FUNCTION_BLOCK FB_MachineControl EXTENDS FB_UniversalMachine IMPLEMENTS I_MachineControl
VAR
	(* Auxilary *)
	iLoop 			: USINT;	
	tonDelay		: TON;			(* Provides any delay into the machine when switching something On/Off *)

	(* --- Sample actuators - from shell template --- DELETE IF NOT NEEDED - *)
	//arrDigitalInput		: ARRAY[0..19] OF FB_DigitalInput;							(* Array of sample digital inputs *)
	//arrDigitalOutput	: ARRAY[0..19] OF FB_DigitalOutput;								(* Array of sample digital outputs *)
	//arrCylinderDc		: ARRAY[0..9] OF FB_DoubleCoilCylinder;							(* Array of sample double coil cylinders *)
	//arrCylinderSc		: ARRAY[0..9] OF FB_SingleCoilCylinder;							(* Array of sample single coil cylinders *)
	//arrAxis				: ARRAY[0..19] OF FB_AxisServo;								(* Array of sample axis *)
	arrRobot			: ARRAY[0..iNUMBER_OF_ROBOTS-1] OF FB_CR800EtherCAT;			(* Array of sample robots *)
	
	tonTestDelay	: TON;	(* Delay which allows to see any page changes during tests *)
	
	(* --- Sample actuators - from shell template --- DELETE IF NOT NEEDED - *)	
	bStart			: BOOL;
	
	(* #ManualToAuto *)             	                                                            		
	bManualToAutoRotate					: BOOL;																            	
	bStop								: BOOL;			
	
	(* CR800 - testing *)
	lrPositionX1 : LREAL := 203.733;
	lrPositionY1 : LREAL := 100.000;
	lrRotation1  : LREAL := 216.699;
	
	lrPositionX2 : LREAL := -13.733;
	lrPositionY2 : LREAL := 8.001;
	lrRotation2  : LREAL := -2.889;
	
	
	bUserDefinedArea1	: BOOL;
	bTryIt1				: BOOL;
	bTryIt2				: BOOL;
	
	(* CR800 EtherCAT diagnostic *) 	                                                                
	fbGetCR800EcState				:  FB_EcGetSlaveState;		
	fbSetCR800CtrlState 			:  FB_EcReqSlaveState;		
	stCR800GetEcState				:  ST_EcSlaveState;		
	
	(* Robots EtherCAT communication *)                      		
	sPLC_NET_ID 							: T_AmsNetId := '5.127.48.8.2.1'; //hardware config							
	iCR800_1_ADDRESS						: UINT	:= 1003; //hardware config										
	//iCR800_2_ADDRESS						: UINT	:= 1016; //hardware config
	
	(* State machines *)	
	eMachineStateUninitialized						: E_MachineCtrlStateUninitialized;
	eMachineStateInit								: E_MachineCtrlStateInit;
	eMachineStateAuto								: E_MachineCtrlStateAuto;
	eMachineStateAutoAOI							: E_MachineCtrlStateAutoAOI;
	eMachineStateAbort								: E_MachineCtrlStateAbort;
	eMachineStateManualToAuto						: E_MachineCtrlStateManualToAuto;
	
END_VAR

IF bFirstCycle THEN
	(* bFirstCycle bit reset by parent *)
	(* --- Assign initial parameters for machine objects ---*)
	(* ---- DELETE IF NOT NEEDED ---- *)
	(* Assign sample robots *)
	FOR iLoop := 0 TO iNUMBER_OF_ROBOTS-1 DO
		arrRobot[iLoop].MR_FirstCycle(	sName		:= CONCAT('Robot_',USINT_TO_STRING(iLoop+1)),
										iOverride	:= 10);
	END_FOR
	(* ---- DELETE IF NOT NEEDED ---- *)
END_IF

(* Execute parent implementation *)
SUPER^();

(* --- Cyclic run of internal objects ---*)
(* Cyclic run of sample robots *)
FOR iLoop := 0 TO iNUMBER_OF_ROBOTS-1 DO
	arrRobot[iLoop]();
END_FOR

//IF bTryIt1 THEN
//	arrRobot[0].MR_SendPosition1( lrPositionX1 := lrPositionX1,
//								lrPositionY1 := lrPositionY1,
//								lrRotation1  := lrRotation1);
//	IF NOT arrRobot[0].SendingPosition1 THEN
//		bTryIt1 := FALSE;
//	END_IF
//END_IF

//IF bTryIt2 THEN
//	arrRobot[0].MR_SendPosition2( lrPositionX2 := lrPositionX2,
//								lrPositionY2 := lrPositionY2,
//								lrRotation2  := lrRotation2);
//	IF NOT arrRobot[0].SendingPosition2 THEN
//		bTryIt1 := FALSE;
//	END_IF
//END_IF

//bUserDefinedArea1 := arrRobot[0].UserDefinedArea1;

tonTestDelay();
(* ---- DELETE IF NOT NEEDED ---- *)

METHOD PRIVATE M_AutoAOI
CASE eMachineStateAutoAOI OF
	MACHINE_STATE_AUTO_AOI_IDLE:
		;
		
	MACHINE_STATE_AUTO_AOI_PROCCESSING:
		eMachineStateAutoAOI := MACHINE_STATE_AUTO_AOI_GO_INPUT;
	
	MACHINE_STATE_AUTO_AOI_GO_INPUT:
		arrRobot[0].ActionNumber := FCQ_ROBOT_ACTION_GO_TO_GS_HIGH_1;
		arrRobot[0].MR_DoAction(iActionNumber := arrRobot[0].ActionNumber);
		IF NOT arrRobot[0].Busy THEN
			eMachineStateAutoAOI := MACHINE_STATE_AUTO_AOI_GO_BACK;
		END_IF		
		
	MACHINE_STATE_AUTO_AOI_GO_BACK:
		arrRobot[0].ActionNumber := FCQ_ROBOT_ACTION_GO_TO_GS_HIGH_2;
		arrRobot[0].MR_DoAction(iActionNumber := arrRobot[0].ActionNumber);
		IF NOT arrRobot[0].Busy THEN
			eMachineStateAutoAOI := MACHINE_STATE_AUTO_AOI_DONE;
		END_IF	
	
	MACHINE_STATE_AUTO_AOI_DONE:
		eMachineStateAutoAOI := MACHINE_STATE_AUTO_AOI_IDLE;
		eMachineStateAuto := MACHINE_STATE_AUTO_IDLE;
END_CASE
END_METHOD

METHOD MR_Start : BOOL
//bRunning := TRUE;

//IF NOT bStart THEN
//	fbMsgAutoStarted.Send(0);
//	bStart := TRUE;
//END_IF

fbMsgAutoStarted.Send(0);

IF eMachineStateAuto = MACHINE_STATE_AUTO_IDLE THEN
	eMachineState := MACHINE_STATE_AUTO;
	eMachineStateAuto := MACHINE_STATE_AUTO_RUNNING;
	
	bStop := FALSE;
	eMachineStateAutoAOI := MACHINE_STATE_AUTO_AOI_PROCCESSING;
END_IF

MR_Start := TRUE;
END_METHOD

METHOD MR_Stop : BOOL
VAR_INPUT
END_VAR
bRunning := FALSE;

IF bStart THEN
	fbMsgAutoStopped.Send(0);
	bStart := FALSE;
END_IF
END_METHOD

METHOD PROTECTED MS_Aborting
(* 
Add here code to abort all machine objects's e.g robots, axes, cylinders. 
At the end add "eMachineState := MACHINE_STATE_UNINITIALIZED;" to finish aborting.
*)
CASE eMachineStateAbort OF
	MACHINE_STATE_ABORTING_ROBOT_CYCLE_STOP:
		arrRobot[0].MR_CycleStop();
		IF arrRobot[0].ErrorOccuring THEN
			arrRobot[0].MR_Init();
		END_IF
		IF NOT arrRobot[0].Busy THEN
			eMachineState := MACHINE_STATE_UNINITIALIZED;
			//eMachineStateAbort := MACHINE_STATE_ABORTING_SAFETY_STOP;
			eMachineStateUninitialized := MACHINE_STATE_UNINITIALIZED_DONE;
		END_IF
END_CASE
END_METHOD

METHOD PROTECTED MS_Auto
CASE eMachineStateAuto OF
	MACHINE_STATE_AUTO_IDLE:
		bRunning := FALSE;
		
	MACHINE_STATE_AUTO_RUNNING:
		bRunning := TRUE;
		M_AutoAOI();
		
END_CASE
END_METHOD

METHOD PROTECTED MS_AutoToManual
VAR_INPUT
END_VAR
(* 
Add here code to switch machine into manual mode. 
At the end add "eMachineState := MACHINE_STATE_MANUAL;" to finish switching.
*)
(* Switching mode to manual simulation - DELETE *)
tonTestDelay(IN := TRUE, PT:= T#500MS);
bRunning := FALSE;
IF tonTestDelay.Q THEN
	tonTestDelay(IN := FALSE);
	eMachineState := MACHINE_STATE_MANUAL;
END_IF
END_METHOD

METHOD PROTECTED MS_Emergency
VAR_INPUT
END_VAR
END_METHOD

METHOD PROTECTED MS_Initializing
(* 
Add here code to initialize all machine objects's e.g robots, axes, cylinders. 
At the end add "eMachineState := MACHINE_STATE_READY_INITIALIZED;" to finish initialization.
*)
CASE eMachineStateInit OF
	MACHINE_STATE_INITIALIZING_MACHINE_LOGGER:
		fbMachineLogger.MR_Init();
		IF NOT fbMachineLogger.Busy THEN
			eMachineStateInit := MACHINE_STATE_INITIALIZING_ROBOTS_POWER_CHECK;
		END_IF
	
	MACHINE_STATE_INITIALIZING_ROBOTS_POWER_CHECK:
		IF arrRobot[0].CR800PoweredOn THEN
			eMachineStateInit := MACHINE_STATE_INITIALIZING_ROBOT_CONTROLERS_RESET;
		END_IF
		
	MACHINE_STATE_INITIALIZING_ROBOT_CONTROLERS_RESET:
		tonDelay( IN := TRUE, PT := T#4S);
		IF tonDelay.Q THEN
			arrRobot[0].MR_ResetCR800Err();			
			IF NOT arrRobot[0].Busy THEN
				tonDelay(IN := FALSE);
				eMachineStateInit := MACHINE_STATE_INITIALIZING_ROBOT_ABORT;
			END_IF
		END_IF
		
	MACHINE_STATE_INITIALIZING_ROBOT_ABORT:
		arrRobot[0].MR_Abort();
		IF NOT arrRobot[0].Active THEN
			eMachineStateInit := MACHINE_STATE_INITIALIZING_ROBOT_INIT;
		END_IF
		
	MACHINE_STATE_INITIALIZING_ROBOT_INIT:
		arrRobot[0].MR_Init();
		IF arrRobot[0].Active THEN
			eMachineStateInit := MACHINE_STATE_INITIALIZING_ROBOT_HOME;
		END_IF
		
	MACHINE_STATE_INITIALIZING_ROBOT_HOME:
		arrRobot[0].MR_GoHome();
		IF NOT arrRobot[0].Busy THEN
			eMachineStateInit := MACHINE_STATE_INITIALIZING_ROBOT_AUTOMATIC_MODE;
		END_IF
		
	MACHINE_STATE_INITIALIZING_ROBOT_AUTOMATIC_MODE:
		arrRobot[0].MR_GoAuto();
		IF NOT arrRobot[0].Busy THEN
			eMachineStateInit := MACHINE_STATE_INITIALIZING_DONE;
		END_IF
		
	MACHINE_STATE_INITIALIZING_DONE:
		eMachineStateInit := MACHINE_STATE_INITIALIZING_MACHINE_LOGGER;
		eMachineState := MACHINE_STATE_READY_INITIALIZED;
END_CASE
END_METHOD

METHOD PROTECTED MS_Manual
VAR_INPUT
END_VAR
(* 
Leave empty - manual mode is provided by HMI controler and automatic frame generator.
*)
;
END_METHOD

METHOD PROTECTED MS_ManualToAuto
VAR_INPUT
END_VAR
(* 
Add here code to switch machine into auto mode. 
At the end add "eMachineState := MACHINE_STATE_AUTO;" to finish switching.
*)
CASE eMachineStateManualToAuto OF
	MACHINE_STATE_MANUAL_TO_AUTO_ROBOT_CYCLE_STOP:
		IF arrRobot[0].ErrorOccuring THEN
			eMachineStateManualToAuto := MACHINE_STATE_MANUAL_TO_AUTO_ROBOT_ABORT;
		ELSE
			arrRobot[0].MR_CycleStop();
			IF NOT arrRobot[0].Busy THEN
				eMachineStateManualToAuto := MACHINE_STATE_MANUAL_TO_AUTO_ROBOT_ABORT;
			END_IF
		END_IF
		
	MACHINE_STATE_MANUAL_TO_AUTO_ROBOT_ABORT:
		arrRobot[0].MR_Abort();
		IF NOT arrRobot[0].Active THEN
			//eMachineStateManualToAuto := MACHINE_STATE_MANUAL_TO_AUTO_ROBOT_REMOTE_MODE;
			eMachineStateManualToAuto := MACHINE_STATE_MANUAL_TO_AUTO_ROBOT_INIT;
		END_IF
	
//	MACHINE_STATE_MANUAL_TO_AUTO_ROBOT_REMOTE_MODE:
//		poRobotModeSwitch.Out := TRUE;
//		tonDelay( IN := TRUE, PT:= T#500MS);
//		IF tonDelay.Q THEN
//			tonDelay(IN := FALSE);
//			eMachineStateManualToAuto := MACHINE_STATE_MANUAL_TO_AUTO_ROBOT_ONE_INIT;
//		END_IF
		
	MACHINE_STATE_MANUAL_TO_AUTO_ROBOT_INIT:
		arrRobot[0].MR_Init();
		IF arrRobot[0].Active THEN
			eMachineStateManualToAuto := MACHINE_STATE_MANUAL_TO_AUTO_ROBOT_HOME;
		END_IF
		
	MACHINE_STATE_MANUAL_TO_AUTO_ROBOT_HOME:
		arrRobot[0].MR_GoHome();
		IF NOT arrRobot[0].Busy THEN
			eMachineStateManualToAuto := MACHINE_STATE_MANUAL_TO_AUTO_ROBOT_AUTOMATIC_MODE;
		END_IF
		
	MACHINE_STATE_MANUAL_TO_AUTO_ROBOT_AUTOMATIC_MODE:
		arrRobot[0].MR_GoAuto();
		IF NOT arrRobot[0].Busy THEN
			eMachineStateManualToAuto := MACHINE_STATE_MANUAL_TO_AUTO_DONE;
		END_IF
		
	MACHINE_STATE_MANUAL_TO_AUTO_DONE:
		eMachineStateManualToAuto := MACHINE_STATE_MANUAL_TO_AUTO_ROBOT_CYCLE_STOP;
		eMachineState := MACHINE_STATE_AUTO;
		
END_CASE
END_METHOD

METHOD PROTECTED MS_ReadyInitialized
VAR_INPUT
END_VAR
(*
Add code here if some internal parameters are needed to set after initialization or leave it default.
At the end add "eMachineState := MACHINE_STATE_AUTO;" to finish and go to IDLE state.
*)
(* Ready-Initialized simulation - DELETE  *)
tonTestDelay(IN := TRUE, PT:= T#500MS);
IF tonTestDelay.Q THEN
	tonTestDelay(IN := FALSE);
	eMachineState := MACHINE_STATE_AUTO;
END_IF
END_METHOD

METHOD PROTECTED MS_Reset
VAR_INPUT
END_VAR
(* 
Add here code to reset all machine objects's e.g robots, axes, cylinders. 
At the end add "eMachineState := MACHINE_STATE_RESET_DONE;" to finish reseting.
*)
(* Reset simulation - DELETE  *)
tonTestDelay(IN := TRUE, PT:= T#4S);
IF tonTestDelay.Q THEN
	tonTestDelay(IN := FALSE);
	eMachineState := MACHINE_STATE_RESET_DONE;
END_IF
END_METHOD

METHOD PROTECTED MS_ResetDone
VAR_INPUT
END_VAR
eMachineState := eMachineStateBeforeReset;
END_METHOD

METHOD PROTECTED MS_Uninitialized
CASE eMachineStateUninitialized OF
	MACHINE_STATE_UNINITIALIZED_CR800_ETHERCAT_STATUS_CHECK:
		fbGetCR800EcState(			sNetId 		:= sPLC_NET_ID,
									nSlaveAddr	:= iCR800_1_ADDRESS,
									bExecute	:= TRUE,
									tTimeout 	:= DEFAULT_ADS_TIMEOUT,
									state		=> stCR800GetEcState);
		IF NOT fbGetCR800EcState.bBusy AND NOT fbGetCR800EcState.bError THEN
			fbGetCR800EcState(bExecute := FALSE);
			eMachineStateUninitialized := MACHINE_STATE_UNINITIALIZED_CR800_ETHERCAT_STATUS_CHECK_DONE;
		END_IF
	
	MACHINE_STATE_UNINITIALIZED_CR800_ETHERCAT_STATUS_CHECK_DONE:
		IF stCR800GetEcState.deviceState = EC_DEVICE_STATE_ERROR OR stCR800GetEcState.deviceState = 84 THEN
			eMachineStateUninitialized := MACHINE_STATE_UNINITIALIZED_CR800_ETHERCAT_ERROR_RESET;
			
		ELSIF stCR800GetEcState.deviceState = EC_DEVICE_STATE_SAFEOP THEN
			eMachineStateUninitialized := MACHINE_STATE_UNINITIALIZED_CR800_ETHERCAT_REQUEST_OP_STATE;
			
		ELSIF stCR800GetEcState.deviceState = EC_DEVICE_STATE_OP THEN
			eMachineStateUninitialized := MACHINE_STATE_UNINITIALIZED_CR800_CHECK_POWER_REGISTER;		
		ELSE
			eMachineStateUninitialized := MACHINE_STATE_UNINITIALIZED_CR800_ETHERCAT_STATUS_CHECK;
		END_IF
		
	MACHINE_STATE_UNINITIALIZED_CR800_ETHERCAT_ERROR_RESET:
		fbSetCR800CtrlState( 		sNetId 		:= sPLC_NET_ID,
									nSlaveAddr	:= iCR800_1_ADDRESS,
									bExecute 	:= TRUE,
									tTimeout 	:= DEFAULT_ADS_TIMEOUT,
									state 		:= EC_DEVICE_STATE_ERROR);
		IF NOT fbSetCR800CtrlState.bBusy AND NOT fbSetCR800CtrlState.bError THEN
			fbSetCR800CtrlState(bExecute := FALSE);
			eMachineStateUninitialized := MACHINE_STATE_UNINITIALIZED_CR800_ETHERCAT_STATUS_CHECK;
		END_IF
		
	MACHINE_STATE_UNINITIALIZED_CR800_ETHERCAT_REQUEST_OP_STATE:
		fbSetCR800CtrlState( 		sNetId 		:= sPLC_NET_ID,
									nSlaveAddr	:= iCR800_1_ADDRESS,
									bExecute 	:= TRUE,
									tTimeout 	:= DEFAULT_ADS_TIMEOUT,
									state 		:= EC_DEVICE_STATE_OP);
		IF NOT fbSetCR800CtrlState.bBusy AND NOT fbSetCR800CtrlState.bError THEN
			fbSetCR800CtrlState(bExecute := FALSE);
			eMachineStateUninitialized := MACHINE_STATE_UNINITIALIZED_CR800_ETHERCAT_STATUS_CHECK;
		END_IF
		
	MACHINE_STATE_UNINITIALIZED_CR800_CHECK_POWER_REGISTER:
		IF arrRobot[0].CR800PoweredOn THEN
			eMachineStateUninitialized := MACHINE_STATE_UNINITIALIZED_DONE;
		END_IF
		
	MACHINE_STATE_UNINITIALIZED_DONE:
		eMachineStateInit := MACHINE_STATE_INITIALIZING_MACHINE_LOGGER;
END_CASE
END_METHOD

PROPERTY Robots : REFERENCE TO ARRAY[0..iNUMBER_OF_ROBOTS-1] OF FB_CR800EtherCAT
GET
Robots REF= arrRobot;
END_GET
END_PROPERTY

PROPERTY StateInit : REFERENCE TO E_MachineCtrlStateInit
GET
StateInit REF= eMachineStateInit;
END_GET
END_PROPERTY

PROPERTY StateUninitialized : REFERENCE TO E_MachineCtrlStateUninitialized
GET
StateUninitialized REF= eMachineStateUninitialized;
END_GET
END_PROPERTY

END_FUNCTION_BLOCK

(* stored: Version 1.1.0.1, ProductVersion 3.1.4024.9
   POU FB_MachineControl: Id {1bd260d7-05fe-41ba-a15a-413659f72f18}, SpecialFunc None
   Folder Internal: Id {8813ce70-337e-4483-a711-2856365d1cdf}
   Folder Properties: Id {29045f01-2b67-43ea-acd9-915a07c376fa}
   Folder Status: Id {971e8d7d-8ce9-4462-b8de-cc46e6b1a59b}
   Folder Requests: Id {51769c61-8807-4a83-b47d-198fbacbeb51}
   Folder StateMachine: Id {fcf2a465-15e6-47fd-a8c6-b9a7900c636c}
   Method M_AutoAOI: Id {5a5cfc22-ae7c-4ab1-a691-e2edd1a85353}
   Method MR_Start: Id {443146db-305a-4222-b20b-6401a2c51521}
   Method MR_Stop: Id {45cc0441-f143-4822-b8f2-bcf21d8684b1}
   Method MS_Aborting: Id {7adc3704-59d9-4656-ad31-e25e008f0070}
   Method MS_Auto: Id {9e955c8e-36bd-49e5-a90f-5a0d0edfdf23}
   Method MS_AutoToManual: Id {02d651de-fd64-4bdf-b695-c41b74db33a4}
   Method MS_Emergency: Id {c21af5de-909a-4da8-88d8-257151739074}
   Method MS_Initializing: Id {99a096da-f0d2-4fb3-bcd1-503614bc69d3}
   Method MS_Manual: Id {cfd995b2-d987-47aa-9bb0-1eb8959a8269}
   Method MS_ManualToAuto: Id {bd4c4af3-faf6-45ca-bf78-e8f80721fb97}
   Method MS_ReadyInitialized: Id {b9fb0eda-7ebb-49ea-ace1-57e0fa237813}
   Method MS_Reset: Id {286f95b6-9876-40be-8c77-b17b043cf4d5}
   Method MS_ResetDone: Id {a6caa836-92e0-4931-80a7-2c291a5ebdf0}
   Method MS_Uninitialized: Id {e7564050-17cc-4cfd-9d7a-3500c05b04b7}
   Property Robots: Id {7f945cab-fcf4-42ea-a55f-ae8887eca31e}
   Get Get: Id {da0b5682-da4c-45e1-aecb-4ccc22637b3c}
   Property StateInit: Id {6264ac4e-9149-4997-8345-6779a81ba273}
   Get Get: Id {f3ca5a5b-5318-49aa-b6c3-043b3b74f2e2}
   Property StateUninitialized: Id {ee5f5748-2f92-4c32-baec-09ffa187a7c0}
   Get Get: Id {5f74a4e1-c4bf-4cc8-9020-607d10150e57} *)
